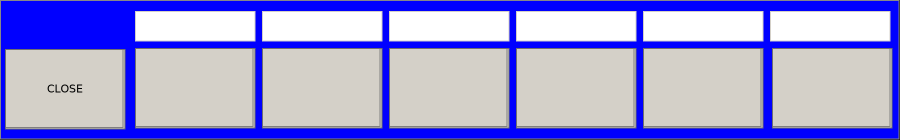
VISUALIZATION dialogStation  // 900x140
    Rectangle (0,0 900x140)
    Group (5,11 887x118)
        Textfield (130,0 120x30), invisible if: NOT gHMIData.gStationEnabled[1], text list: 'ModeStates', text index: S1_Global.station.Data.StationState
        Textfield (257,0 120x30), invisible if: NOT gHMIData.gStationEnabled[2], text list: 'ModeStates', text index: S2_Global.station.Data.StationState
        Textfield (384,0 120x30), invisible if: NOT gHMIData.gStationEnabled[3], text list: 'ModeStates', text index: S3_Global.station.Data.StationState
        Textfield (511,0 120x30), invisible if: NOT gHMIData.gStationEnabled[4], text list: 'ModeStates', text index: S4_Global.station.Data.StationState
        Textfield (638,0 120x30), invisible if: NOT gHMIData.gStationEnabled[5], text list: 'ModeStates', text index: S5_Global.station.Data.StationState
        Textfield (765,0 120x30), invisible if: NOT gHMIData.gStationEnabled[6], text list: 'ModeStates', text index: S6_Global.station.Data.StationState
        Button (130,37 120x80), colour toggle: gHMIData.gStationSelected[1], invisible if: NOT gHMIData.gStationEnabled[1], text list: 'StationNames', text index: 1
            tap gHMIButtons.btnSelectStation1
            OnMouseClick: CloseDialog Dialog=dialogStation, Result=OK, NumpadKeypadSet=True
        Button (257,37 120x80), colour toggle: gHMIData.gStationSelected[2], invisible if: NOT gHMIData.gStationEnabled[2], text list: 'StationNames', text index: 2
            tap gHMIButtons.btnSelectStation2
            OnMouseClick: CloseDialog Dialog=dialogStation, Result=OK, NumpadKeypadSet=True
        Button (384,37 120x80), colour toggle: gHMIData.gStationSelected[3], invisible if: NOT gHMIData.gStationEnabled[3], text list: 'StationNames', text index: 3
            tap gHMIButtons.btnSelectStation3
            OnMouseClick: CloseDialog Dialog=dialogStation, Result=OK, NumpadKeypadSet=True
        Button (511,37 120x80), colour toggle: gHMIData.gStationSelected[4], invisible if: NOT gHMIData.gStationEnabled[4], text list: 'StationNames', text index: 4
            tap gHMIButtons.btnSelectStation4
            OnMouseClick: CloseDialog Dialog=dialogStation, Result=OK, NumpadKeypadSet=True
        Button (638,37 120x80), colour toggle: gHMIData.gStationSelected[5], invisible if: NOT gHMIData.gStationEnabled[5], text list: 'StationNames', text index: 5
            tap gHMIButtons.btnSelectStation5
            OnMouseClick: CloseDialog Dialog=dialogStation, Result=OK, NumpadKeypadSet=True
        Button (767,37 120x80), colour toggle: gHMIData.gStationSelected[6], invisible if: NOT gHMIData.gStationEnabled[6], text list: 'StationNames', text index: 6
            tap gHMIButtons.btnSelectStation6
            OnMouseClick: CloseDialog Dialog=dialogStation, Result=OK, NumpadKeypadSet=True
        Button (0,38 120x80), "CLOSE", colour toggle: gHMIButtons.btnAllStationsSelected, text list: ''
            OnMouseClick: CloseDialog Dialog=dialogStation, Result=None, NumpadKeypadSet=True
END_VISUALIZATION

(* stored: Version 1.1.0.1, ProductVersion 3.1.4024.12
   Visu dialogStation: Id {d75ffeef-a555-485a-9d1a-0b78789cb753} *)
